{attribute 'qualified_only'}
{attribute 'strict'}
TYPE DUT :
(
	enum_member := 0
);
END_TYPE

(* stored: Version 1.1.0.1, ProductVersion 3.1.4022.10
   EnumerationTextList DUT: Id {ea9d9389-424d-4c27-b743-4e5e048daef5} *)
